FUNCTION_BLOCK EL2634
VAR
	{attribute addProperty Name "WcState"}
	_wcState : WcStateBase;
	{attribute addProperty Name "Info data"}
	_infoData : InfoDataBase;
	_io : EL2xx4_Data;
END_VAR

PROPERTY IO : REFERENCE TO EL2xx4_Data
GET
IO REF= _io;
END_GET
END_PROPERTY

PROPERTY WcState : REFERENCE TO WcStateBase
GET
WcState REF= _wcState;
END_GET
END_PROPERTY

END_FUNCTION_BLOCK

(* stored: Version 1.1.0.1, ProductVersion 3.1.4024.9
   POU EL2634: Id {c754c3cf-2d27-0117-1a73-4969ad0ee0bf}, SpecialFunc None
   Property IO: Id {96ed1ae4-32ca-0b3a-1dd8-6879d324d7a9}
   Get Get: Id {08721272-9bd3-0f43-0849-c52f11f74735}
   Property WcState: Id {2609a48d-90ed-0214-1f84-c4f614866d8b}
   Get Get: Id {9613ea7a-5f2e-09e0-04be-01af96cf0fff} *)
